TYPE ST_FunctionInterfaceIn :
(**************************************************************************************
 * 	Application		:	BoxControl Framework
 *	Revision		:	$Revision: 404529 $
 *	Revision date	:	$Date: 2018-04-23 08:21:38 +0200 (Mo., 23 Apr 2018) $
 *	Last changed by	:	$Author: b7bolm $
 *	URL				:	$URL: http://almscdc.swisslog.com/repo/SWPD/Development/BoxControlFramework/20_Release/trunk/01_Software/BCF/BCF/JumpStart/20_Product/10_App/12_E_Functions/10_Lib/10_Conv/01_DUTs/ST_FunctionInterfaceIn.TcDUT $
 *
 *	Purpose			:	Function interface - Contains data which is provided by the
 *						function or is input from other objects.
 *
 * ------------------------------------------------------------------------------------
 *	Copyright Swisslog [IP AG], Switzerland. All rights reserved.
 * 
 * ------------------------------------------------------------------------------------
 *	
 * 	Revision History: 
 *
 * 	VERSION			DATE			INITIALS			DESCRIPTION
 *	0.1				01.01.2001		swl					Example
 *
 **************************************************************************************)
STRUCT
	ePrevFunctionNumber 	: E_FunctionNumber; // Previous element function number
	eNextFunctionNumber 	: E_FunctionNumber; // Next element function number	
	FunctionEnable			: BOOL := TRUE; // External function enable 
	Element					: ST_FunctionElement; // States of the function corresponding element
	AddOnOrder				: ARRAY [1..Conveyor.NUMBER_OF_ADDON_FUNCTIONS] OF ST_AddOn; // Number of addons per function
END_STRUCT
END_TYPE

(* stored: Version 1.1.0.1, ProductVersion 3.1.4022.12
   DUT ST_FunctionInterfaceIn: Id {7c05c4ca-05e1-4b88-8c3a-3c9756eb4769} *)
